// Bidirectional linear motor
FUNCTION_BLOCK FB_LinearMotor  
VAR_INPUT
	bAlarmSignal: BOOL;        // NC alarm signal from the device
END_VAR
VAR_OUTPUT
	bMoveToPick: BOOL;         // Output for motor to drive forward
	bMoveToPlace: BOOL;        // Output for motor to drive backward
	bError: BOOL;              // Motor is in error
END_VAR
VAR
END_VAR

IF inError THEN                // Stop the motor if it is in th error state
	Stop();        
	bError := TRUE;
ELSE
	bError := FALSE;
END_IF

// Motor is in the error state
PROPERTY inError : Bool
GET
inError := NOT bAlarmSignal; // Motor is in error state when there is no NC alarm signal
END_GET
END_PROPERTY

// Move to the pick position
METHOD MoveToPick : BOOL

VAR_INPUT

END_VAR
bMoveToPick := TRUE;   // Set output for motor to drive forward
bMoveToPlace:= FALSE;  // Reset output for motor to drive backward
END_METHOD

// Move to the place position
METHOD MoveToPlace : BOOL
VAR_INPUT
END_VAR
bMoveToPick := FALSE;  // Reset output for motor to drive forward
bMoveToPlace:= TRUE;   // Set output for motor to drive backward
END_METHOD

// Stop the motor 
METHOD Stop : BOOL
VAR_INPUT
END_VAR
bMoveToPick := FALSE;  // Reset output for motor to drive forward
bMoveToPlace:= FALSE;  // Reset output for motor to drive backward
END_METHOD

END_FUNCTION_BLOCK

(* stored: Version 1.1.0.1, ProductVersion 3.1.4024.12
   POU FB_LinearMotor: Id {6f182d56-d000-45d3-8927-eedc37f7075e}, SpecialFunc None
   Property inError: Id {8f2295b2-2df4-42c2-938f-27eb134e2997}
   Get Get: Id {b88da420-2e86-42b1-b6b6-b1b510ba97ab}
   Method MoveToPick: Id {ba39bd66-f20f-43ca-a17f-8f0430306b55}
   Method MoveToPlace: Id {5a65e9de-c118-4280-b8a0-9c384f9af79a}
   Method Stop: Id {0f166531-81c2-4645-91a9-e231ac44df24} *)
